TYPE ST_MasterAxis :
STRUCT
	i		:	UINT:=1;	//Master axis index
	ratio	:	LREAL;	//Gear Ratio
END_STRUCT
END_TYPE

(* stored: Version 1.1.0.1, ProductVersion 3.1.4022.12
   DUT ST_MasterAxis: Id {14b8b990-f919-41af-832a-7d1ca130ac78} *)
